(* 
:Description: This function block takes care of persistent data save for 1 second UPS from CX51xx series 
*)
FUNCTION_BLOCK FB_UpsCx51xx EXTENDS FB_UpsCx5xxx
VAR
	fbSavePersistentData : FB_S_UPS_CX51x0;	(*  *)
END_VAR
(*
Version history:

+-------------+------------+----------------+----------+------------------------------------------+
|Date         | Version    | created under  | Author   | Remark                                   |
+=============+============+================+==========+==========================================+
|2021-11      | 1.0.0.0    | V3.1.4024.22   | ADBO     | Function block created                   |
+-------------+------------+----------------+----------+------------------------------------------+
|2022-01      | 1.1.0.0    | V3.1.4024.22   | ADBO     | Changed to extension of FB_UpsCx5xxx     |
+-------------+------------+----------------+----------+------------------------------------------+

*)

IF bFirstCycle THEN
	bFirstCycle := FALSE;
	iUpsPort := 16#588;
END_IF

(* Save persistent data when an power failure occurred *)
fbSavePersistentData(	sNetID			:= sNetID,
						iPLCPort		:= iPlcPort,
						iUPSPort		:= iUpsPort,
						tTimeout		:= tTimeout,
						eUpsMode		:= eUpsMode,
						ePersistentMode	:= ePersistentMode,
						tRecoverTime 	:= tRecoverTime);

bPowerOk := NOT fbSavePersistentData.bPowerFailDetect;

END_FUNCTION_BLOCK

(* stored: Version 1.1.0.1, ProductVersion 3.1.4024.12
   POU FB_UpsCx51xx: Id {8ae3296f-f5a5-4c78-8bce-e1d60466ccdc}, SpecialFunc None *)
